FUNCTION_BLOCK gabriel_xor
  (* Standard: 61499-2 *)
  (* Version 11-01-12, GASR *)
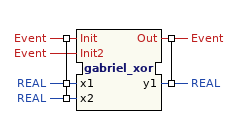
  EVENT_INPUT
    Init WITH x1, x2;
    Init2;
  END_EVENT
  EVENT_OUTPUT
    Out WITH y1;
  END_EVENT
  VAR_INPUT
    x1 : REAL;
    x2 : REAL;
  END_VAR
  VAR_OUTPUT
    y1 : REAL;
  END_VAR
END_FUNCTION_BLOCK
